{attribute 'qualified_only'}
VAR_GLOBAL
  Com : ZCom;
END_VAR
VAR_GLOBAL PERSISTENT
  Data : ZData;
END_VAR

(* stored: Version 1.1.0.1
   GVL ZGlobal: Id {bea27b08-115f-4b55-bfcb-764f02427eee} *)
